// TIA Portal V20 export
DATA_BLOCK "Config"   // DB58
{ DB_Accessible_From_OPC_UA := 'FALSE' }
AUTHOR : ERsystem_FA2_DH. Kim
// stored: Access Published, DBAccessibleFromOPCUA false, DBAccessibleFromWebserver false, MemoryReserve 100, Namespace Unit1.Em6
   VAR
      em { ExternalWritable := 'False'} : "LAF_typeEmConfiguration";
      axis { ExternalAccessible := 'False'; ExternalVisible := 'False'; ExternalWritable := 'False'} : Array[1.._.U1EM6_NO_OF_AXES] of DB_ANY;
      outputCam : Array[1.._.U1EM6_NO_OF_OUTPUTCAM] of DB_ANY;
      cmStackTableElectrodeDetect { S7_SetPoint := 'True'} : "LBC_typeDigitalSignalConfiguration";
   END_VAR
   VAR RETAIN
      cmMasterVirtualAxisX { ExternalVisible := 'False'; ExternalWritable := 'False'} : "LBC_typeAxis64PosConfiguration";
      cmFinalRollerFrontAxisX { ExternalVisible := 'False'; ExternalWritable := 'False'} : "LBC_typeAxis64PosConfiguration";
      cmFinalRollerRearAxisX { ExternalVisible := 'False'; ExternalWritable := 'False'; S7_SetPoint := 'True'} : "LBC_typeAxis64PosConfiguration";
      cmMendrelAnodeFrontAxisY { ExternalVisible := 'False'; ExternalWritable := 'False'; S7_SetPoint := 'True'} : "LBC_typeAxis64PosConfiguration";
      cmMendrelAnodeFrontAxisZ { ExternalVisible := 'False'; ExternalWritable := 'False'; S7_SetPoint := 'True'} : "LBC_typeAxis64PosConfiguration";
      cmMendrelAnodeRearAxisY { ExternalVisible := 'False'; ExternalWritable := 'False'; S7_SetPoint := 'True'} : "LBC_typeAxis64PosConfiguration";
      cmMendrelAnodeRearAxisZ { ExternalVisible := 'False'; ExternalWritable := 'False'; S7_SetPoint := 'True'} : "LBC_typeAxis64PosConfiguration";
      cmMendrelCathodeFrontAxisY { ExternalVisible := 'False'; ExternalWritable := 'False'; S7_SetPoint := 'True'} : "LBC_typeAxis64PosConfiguration";
      cmMendrelCathodeFrontAxisZ { ExternalVisible := 'False'; ExternalWritable := 'False'; S7_SetPoint := 'True'} : "LBC_typeAxis64PosConfiguration";
      cmMendrelCathodeRearAxisY { ExternalVisible := 'False'; ExternalWritable := 'False'; S7_SetPoint := 'True'} : "LBC_typeAxis64PosConfiguration";
      cmMendrelCathodeRearAxisZ { ExternalVisible := 'False'; ExternalWritable := 'False'; S7_SetPoint := 'True'} : "LBC_typeAxis64PosConfiguration";
      cmStackTableAxisZ { ExternalVisible := 'False'; ExternalWritable := 'False'; S7_SetPoint := 'True'} : "LBC_typeAxis64PosConfiguration";
      cmStackTableOutFrontAxisZ { ExternalVisible := 'False'; ExternalWritable := 'False'; S7_SetPoint := 'True'} : "LBC_typeAxis64PosConfiguration";
      cmStackTableOutRearAxisZ { ExternalVisible := 'False'; ExternalWritable := 'False'; S7_SetPoint := 'True'} : "LBC_typeAxis64PosConfiguration";
   END_VAR
   VAR
      cmMendrelAnodeFrontClamp { ExternalAccessible := 'False'; ExternalVisible := 'False'; ExternalWritable := 'False'; S7_SetPoint := 'True'} : "LBC_typeTwoWayActuatorConfiguration";
      cmMendrelAnodeRearClamp { ExternalAccessible := 'False'; ExternalVisible := 'False'; ExternalWritable := 'False'; S7_SetPoint := 'True'} : "LBC_typeTwoWayActuatorConfiguration";
      cmMendrelCathodeFrontClamp { ExternalAccessible := 'False'; ExternalVisible := 'False'; ExternalWritable := 'False'; S7_SetPoint := 'True'} : "LBC_typeTwoWayActuatorConfiguration";
      cmMendrelCathodeRearClamp { ExternalAccessible := 'False'; ExternalVisible := 'False'; ExternalWritable := 'False'; S7_SetPoint := 'True'} : "LBC_typeTwoWayActuatorConfiguration";
      cmStackTableVaccum { ExternalAccessible := 'False'; ExternalVisible := 'False'; ExternalWritable := 'False'; S7_SetPoint := 'True'} : "LBC_typeTwoWayActuatorConfiguration";
      cmStackTableGapPadUpDown { ExternalAccessible := 'False'; ExternalVisible := 'False'; ExternalWritable := 'False'; S7_SetPoint := 'True'} : "LBC_typeTwoWayActuatorConfiguration";
      cmStackGapVisionControllerInterface { ExternalAccessible := 'False'; ExternalVisible := 'False'; ExternalWritable := 'False'; S7_SetPoint := 'True'} : "LER_typeVisionConfiguration";
   END_VAR
   VAR RETAIN
      softCam : Struct
         cmFinalRollerFrontAxisX : "LER_typeSoftCamInterface";
         cmFinalRollerRearAxisX { S7_SetPoint := 'True'} : "LER_typeSoftCamInterface";
         cmMendrelAnodeFrontAxisY { S7_SetPoint := 'True'} : "LER_typeSoftCamInterface";
         cmMendrelAnodeFrontAxisZ { S7_SetPoint := 'True'} : "LER_typeSoftCamInterface";
         cmMendrelAnodeRearAxisY { S7_SetPoint := 'True'} : "LER_typeSoftCamInterface";
         cmMendrelAnodeRearAxisZ { S7_SetPoint := 'True'} : "LER_typeSoftCamInterface";
         cmMendrelCathodeFrontAxisY { S7_SetPoint := 'True'} : "LER_typeSoftCamInterface";
         cmMendrelCathodeFrontAxisZ { S7_SetPoint := 'True'} : "LER_typeSoftCamInterface";
         cmMendrelCathodeRearAxisY { S7_SetPoint := 'True'} : "LER_typeSoftCamInterface";
         cmMendrelCathodeRearAxisZ { S7_SetPoint := 'True'} : "LER_typeSoftCamInterface";
         cmStackTableAxisZ { S7_SetPoint := 'True'} : "LER_typeSoftCamInterface";
         cmStackTableOutFrontAxisZ { S7_SetPoint := 'True'} : "LER_typeSoftCamInterface";
         cmStackTableOutRearAxisZ { S7_SetPoint := 'True'} : "LER_typeSoftCamInterface";
      END_STRUCT;
   END_VAR
BEGIN
   em.referenceDesignator.parent := WSTRING#'';
   em.referenceDesignator.relative := WSTRING#'';
   em.referenceDesignator.combined := WSTRING#'';
   axis[1] := 171;   // FinalRollerFrontAxisX
   axis[2] := 172;   // FinalRollerRearAxisX
   axis[3] := 163;   // MendrelAnodeFrontAxisY
   axis[4] := 162;   // MendrelAnodeFrontAxisZ
   axis[5] := 167;   // MendrelAnodeRearAxisY
   axis[6] := 166;   // MendrelAnodeRearAxisZ
   axis[7] := 161;   // MendrelCathodeFrontAxisY
   axis[8] := 160;   // MendrelCathodeFrontAxisZ
   axis[9] := 165;   // MendrelCathodeRearAxisY
   axis[10] := 164;   // MendrelCathodeRearAxisZ
   axis[11] := 168;   // StackTableAxisZ
   axis[12] := 169;   // StackTableOutFrontAxisZ
   axis[13] := 170;   // StackTableOutRearAxisZ
   axis[14] := 85;
   outputCam[1] := 224;
   outputCam[2] := 225;
   outputCam[3] := 206;
   outputCam[4] := 446;
   outputCam[5] := 445;
   outputCam[6] := 84;
   cmStackTableElectrodeDetect.referenceDesignator := WSTRING#'DigitalSignal';
   cmStackTableElectrodeDetect.onDelay := T#0MS;
   cmStackTableElectrodeDetect.offDelay := T#0MS;
   cmStackTableElectrodeDetect.default := FALSE;
   cmStackTableElectrodeDetect.invertProcessValue := FALSE;
   cmStackTableElectrodeDetect.disableAlarms := FALSE;
   cmMasterVirtualAxisX.referenceDesignator := WSTRING#'FinalRollerFrontAxisX';
   cmMasterVirtualAxisX.disableAlarms := FALSE;
   cmMasterVirtualAxisX.masterControlPopUp := TRUE;
   cmMasterVirtualAxisX.setPositions[0..15].position := 0.0;
   cmMasterVirtualAxisX.setPositions[0..15].velocity := -1.0;
   cmMasterVirtualAxisX.setPositions[0..15].acceleration := -1.0;
   cmMasterVirtualAxisX.setPositions[0..15].deceleration := -1.0;
   cmMasterVirtualAxisX.setPositions[0..15]."name" := '';
   cmFinalRollerFrontAxisX.referenceDesignator := WSTRING#'FinalRollerFrontAxisX';
   cmFinalRollerFrontAxisX.disableAlarms := FALSE;
   cmFinalRollerFrontAxisX.masterControlPopUp := TRUE;
   cmFinalRollerFrontAxisX.setPositions[0].position := 0.0;
   cmFinalRollerFrontAxisX.setPositions[1].position := 310.0;
   cmFinalRollerFrontAxisX.setPositions[2..15].position := 0.0;
   cmFinalRollerFrontAxisX.setPositions[0..1].velocity := 500.0;
   cmFinalRollerFrontAxisX.setPositions[2..3].velocity := 16#7FF8_0000_0000_0000;
   cmFinalRollerFrontAxisX.setPositions[4..15].velocity := -1.0;
   cmFinalRollerFrontAxisX.setPositions[0..1].acceleration := 5000.0;
   cmFinalRollerFrontAxisX.setPositions[2..3].acceleration := 16#7FF8_0000_0000_0000;
   cmFinalRollerFrontAxisX.setPositions[4..15].acceleration := -1.0;
   cmFinalRollerFrontAxisX.setPositions[0..1].deceleration := 5000.0;
   cmFinalRollerFrontAxisX.setPositions[2..3].deceleration := 16#7FF8_0000_0000_0000;
   cmFinalRollerFrontAxisX.setPositions[4..15].deceleration := -1.0;
   cmFinalRollerFrontAxisX.setPositions[0..15]."name" := '';
   cmFinalRollerRearAxisX.referenceDesignator := WSTRING#'FinalRollerRearAxisX';
   cmFinalRollerRearAxisX.disableAlarms := FALSE;
   cmFinalRollerRearAxisX.masterControlPopUp := TRUE;
   cmFinalRollerRearAxisX.setPositions[0].position := 0.0;
   cmFinalRollerRearAxisX.setPositions[1].position := 310.0;
   cmFinalRollerRearAxisX.setPositions[2..15].position := 0.0;
   cmFinalRollerRearAxisX.setPositions[0..1].velocity := 500.0;
   cmFinalRollerRearAxisX.setPositions[2..3].velocity := 16#7FF8_0000_0000_0000;
   cmFinalRollerRearAxisX.setPositions[4..15].velocity := -1.0;
   cmFinalRollerRearAxisX.setPositions[0..1].acceleration := 5000.0;
   cmFinalRollerRearAxisX.setPositions[2..3].acceleration := 16#7FF8_0000_0000_0000;
   cmFinalRollerRearAxisX.setPositions[4..15].acceleration := -1.0;
   cmFinalRollerRearAxisX.setPositions[0..1].deceleration := 5000.0;
   cmFinalRollerRearAxisX.setPositions[2..3].deceleration := 16#7FF8_0000_0000_0000;
   cmFinalRollerRearAxisX.setPositions[4..15].deceleration := -1.0;
   cmFinalRollerRearAxisX.setPositions[0..15]."name" := '';
   cmMendrelAnodeFrontAxisY.referenceDesignator := WSTRING#'MendrelAnodeFrontAxisY';
   cmMendrelAnodeFrontAxisY.disableAlarms := FALSE;
   cmMendrelAnodeFrontAxisY.masterControlPopUp := TRUE;
   cmMendrelAnodeFrontAxisY.setPositions[0].position := 0.0;
   cmMendrelAnodeFrontAxisY.setPositions[1].position := 50.0;
   cmMendrelAnodeFrontAxisY.setPositions[2..15].position := 0.0;
   cmMendrelAnodeFrontAxisY.setPositions[0..1].velocity := 50.0;
   cmMendrelAnodeFrontAxisY.setPositions[2..15].velocity := -1.0;
   cmMendrelAnodeFrontAxisY.setPositions[0..1].acceleration := 500.0;
   cmMendrelAnodeFrontAxisY.setPositions[2..15].acceleration := -1.0;
   cmMendrelAnodeFrontAxisY.setPositions[0..1].deceleration := 500.0;
   cmMendrelAnodeFrontAxisY.setPositions[2..15].deceleration := -1.0;
   cmMendrelAnodeFrontAxisY.setPositions[0..15]."name" := '';
   cmMendrelAnodeFrontAxisZ.referenceDesignator := WSTRING#'MendrelAnodeFrontAxisZ';
   cmMendrelAnodeFrontAxisZ.disableAlarms := FALSE;
   cmMendrelAnodeFrontAxisZ.masterControlPopUp := TRUE;
   cmMendrelAnodeFrontAxisZ.setPositions[0].position := 0.0;
   cmMendrelAnodeFrontAxisZ.setPositions[1].position := 50.0;
   cmMendrelAnodeFrontAxisZ.setPositions[2..15].position := 0.0;
   cmMendrelAnodeFrontAxisZ.setPositions[0..1].velocity := 50.0;
   cmMendrelAnodeFrontAxisZ.setPositions[2..15].velocity := -1.0;
   cmMendrelAnodeFrontAxisZ.setPositions[0..1].acceleration := 500.0;
   cmMendrelAnodeFrontAxisZ.setPositions[2..15].acceleration := -1.0;
   cmMendrelAnodeFrontAxisZ.setPositions[0..1].deceleration := 500.0;
   cmMendrelAnodeFrontAxisZ.setPositions[2..15].deceleration := -1.0;
   cmMendrelAnodeFrontAxisZ.setPositions[0..15]."name" := '';
   cmMendrelAnodeRearAxisY.referenceDesignator := WSTRING#'MendrelAnodeRearAxisY';
   cmMendrelAnodeRearAxisY.disableAlarms := FALSE;
   cmMendrelAnodeRearAxisY.masterControlPopUp := TRUE;
   cmMendrelAnodeRearAxisY.setPositions[0].position := 0.0;
   cmMendrelAnodeRearAxisY.setPositions[1].position := 50.0;
   cmMendrelAnodeRearAxisY.setPositions[2..15].position := 0.0;
   cmMendrelAnodeRearAxisY.setPositions[0..1].velocity := 50.0;
   cmMendrelAnodeRearAxisY.setPositions[2..15].velocity := -1.0;
   cmMendrelAnodeRearAxisY.setPositions[0..1].acceleration := 500.0;
   cmMendrelAnodeRearAxisY.setPositions[2..15].acceleration := -1.0;
   cmMendrelAnodeRearAxisY.setPositions[0..1].deceleration := 500.0;
   cmMendrelAnodeRearAxisY.setPositions[2..15].deceleration := -1.0;
   cmMendrelAnodeRearAxisY.setPositions[0..15]."name" := '';
   cmMendrelAnodeRearAxisZ.referenceDesignator := WSTRING#'MendrelAnodeRearAxisZ';
   cmMendrelAnodeRearAxisZ.disableAlarms := FALSE;
   cmMendrelAnodeRearAxisZ.masterControlPopUp := TRUE;
   cmMendrelAnodeRearAxisZ.setPositions[0].position := 0.0;
   cmMendrelAnodeRearAxisZ.setPositions[1].position := 50.0;
   cmMendrelAnodeRearAxisZ.setPositions[2..15].position := 0.0;
   cmMendrelAnodeRearAxisZ.setPositions[0..1].velocity := 50.0;
   cmMendrelAnodeRearAxisZ.setPositions[2..15].velocity := -1.0;
   cmMendrelAnodeRearAxisZ.setPositions[0..1].acceleration := 500.0;
   cmMendrelAnodeRearAxisZ.setPositions[2..15].acceleration := -1.0;
   cmMendrelAnodeRearAxisZ.setPositions[0..1].deceleration := 500.0;
   cmMendrelAnodeRearAxisZ.setPositions[2..15].deceleration := -1.0;
   cmMendrelAnodeRearAxisZ.setPositions[0..15]."name" := '';
   cmMendrelCathodeFrontAxisY.referenceDesignator := WSTRING#'MendrelCathodeFrontAxisY';
   cmMendrelCathodeFrontAxisY.disableAlarms := FALSE;
   cmMendrelCathodeFrontAxisY.masterControlPopUp := TRUE;
   cmMendrelCathodeFrontAxisY.setPositions[0].position := 0.0;
   cmMendrelCathodeFrontAxisY.setPositions[1].position := 50.0;
   cmMendrelCathodeFrontAxisY.setPositions[2..15].position := 0.0;
   cmMendrelCathodeFrontAxisY.setPositions[0..1].velocity := 50.0;
   cmMendrelCathodeFrontAxisY.setPositions[2..15].velocity := -1.0;
   cmMendrelCathodeFrontAxisY.setPositions[0..1].acceleration := 500.0;
   cmMendrelCathodeFrontAxisY.setPositions[2..15].acceleration := -1.0;
   cmMendrelCathodeFrontAxisY.setPositions[0..1].deceleration := 500.0;
   cmMendrelCathodeFrontAxisY.setPositions[2..15].deceleration := -1.0;
   cmMendrelCathodeFrontAxisY.setPositions[0..15]."name" := '';
   cmMendrelCathodeFrontAxisZ.referenceDesignator := WSTRING#'MendrelCathodeFrontAxisZ';
   cmMendrelCathodeFrontAxisZ.disableAlarms := FALSE;
   cmMendrelCathodeFrontAxisZ.masterControlPopUp := TRUE;
   cmMendrelCathodeFrontAxisZ.setPositions[0].position := 0.0;
   cmMendrelCathodeFrontAxisZ.setPositions[1].position := 50.0;
   cmMendrelCathodeFrontAxisZ.setPositions[2..15].position := 0.0;
   cmMendrelCathodeFrontAxisZ.setPositions[0..1].velocity := 50.0;
   cmMendrelCathodeFrontAxisZ.setPositions[2..15].velocity := -1.0;
   cmMendrelCathodeFrontAxisZ.setPositions[0..1].acceleration := 500.0;
   cmMendrelCathodeFrontAxisZ.setPositions[2..15].acceleration := -1.0;
   cmMendrelCathodeFrontAxisZ.setPositions[0..1].deceleration := 500.0;
   cmMendrelCathodeFrontAxisZ.setPositions[2..15].deceleration := -1.0;
   cmMendrelCathodeFrontAxisZ.setPositions[0..15]."name" := '';
   cmMendrelCathodeRearAxisY.referenceDesignator := WSTRING#'MendrelCathodeRearAxisY';
   cmMendrelCathodeRearAxisY.disableAlarms := FALSE;
   cmMendrelCathodeRearAxisY.masterControlPopUp := TRUE;
   cmMendrelCathodeRearAxisY.setPositions[0].position := 0.0;
   cmMendrelCathodeRearAxisY.setPositions[1].position := 50.0;
   cmMendrelCathodeRearAxisY.setPositions[2..15].position := 0.0;
   cmMendrelCathodeRearAxisY.setPositions[0..1].velocity := 50.0;
   cmMendrelCathodeRearAxisY.setPositions[2..15].velocity := -1.0;
   cmMendrelCathodeRearAxisY.setPositions[0..1].acceleration := 500.0;
   cmMendrelCathodeRearAxisY.setPositions[2..15].acceleration := -1.0;
   cmMendrelCathodeRearAxisY.setPositions[0..1].deceleration := 500.0;
   cmMendrelCathodeRearAxisY.setPositions[2..15].deceleration := -1.0;
   cmMendrelCathodeRearAxisY.setPositions[0..15]."name" := '';
   cmMendrelCathodeRearAxisZ.referenceDesignator := WSTRING#'MendrelCathodeRearAxisZ';
   cmMendrelCathodeRearAxisZ.disableAlarms := FALSE;
   cmMendrelCathodeRearAxisZ.masterControlPopUp := TRUE;
   cmMendrelCathodeRearAxisZ.setPositions[0].position := 0.0;
   cmMendrelCathodeRearAxisZ.setPositions[1].position := 50.0;
   cmMendrelCathodeRearAxisZ.setPositions[2..15].position := 0.0;
   cmMendrelCathodeRearAxisZ.setPositions[0..1].velocity := 50.0;
   cmMendrelCathodeRearAxisZ.setPositions[2..15].velocity := -1.0;
   cmMendrelCathodeRearAxisZ.setPositions[0..1].acceleration := 500.0;
   cmMendrelCathodeRearAxisZ.setPositions[2..15].acceleration := -1.0;
   cmMendrelCathodeRearAxisZ.setPositions[0..1].deceleration := 500.0;
   cmMendrelCathodeRearAxisZ.setPositions[2..15].deceleration := -1.0;
   cmMendrelCathodeRearAxisZ.setPositions[0..15]."name" := '';
   cmStackTableAxisZ.referenceDesignator := WSTRING#'StackTableAxisZ';
   cmStackTableAxisZ.disableAlarms := FALSE;
   cmStackTableAxisZ.masterControlPopUp := TRUE;
   cmStackTableAxisZ.setPositions[0].position := 0.0;
   cmStackTableAxisZ.setPositions[1].position := 5.0;
   cmStackTableAxisZ.setPositions[2..15].position := 0.0;
   cmStackTableAxisZ.setPositions[0..1].velocity := 50.0;
   cmStackTableAxisZ.setPositions[2..15].velocity := -1.0;
   cmStackTableAxisZ.setPositions[0..1].acceleration := 500.0;
   cmStackTableAxisZ.setPositions[2..15].acceleration := -1.0;
   cmStackTableAxisZ.setPositions[0..1].deceleration := 500.0;
   cmStackTableAxisZ.setPositions[2..15].deceleration := -1.0;
   cmStackTableAxisZ.setPositions[0..15]."name" := '';
   cmStackTableOutFrontAxisZ.referenceDesignator := WSTRING#'StackTableOutFrontAxisZ';
   cmStackTableOutFrontAxisZ.disableAlarms := FALSE;
   cmStackTableOutFrontAxisZ.masterControlPopUp := TRUE;
   cmStackTableOutFrontAxisZ.setPositions[0].position := 0.0;
   cmStackTableOutFrontAxisZ.setPositions[1].position := 500.0;
   cmStackTableOutFrontAxisZ.setPositions[2..15].position := 0.0;
   cmStackTableOutFrontAxisZ.setPositions[0..1].velocity := 500.0;
   cmStackTableOutFrontAxisZ.setPositions[2..15].velocity := -1.0;
   cmStackTableOutFrontAxisZ.setPositions[0..1].acceleration := 5000.0;
   cmStackTableOutFrontAxisZ.setPositions[2..15].acceleration := -1.0;
   cmStackTableOutFrontAxisZ.setPositions[0..1].deceleration := 5000.0;
   cmStackTableOutFrontAxisZ.setPositions[2..15].deceleration := -1.0;
   cmStackTableOutFrontAxisZ.setPositions[0..15]."name" := '';
   cmStackTableOutRearAxisZ.referenceDesignator := WSTRING#'StackTableOutRearAxisZ';
   cmStackTableOutRearAxisZ.disableAlarms := FALSE;
   cmStackTableOutRearAxisZ.masterControlPopUp := TRUE;
   cmStackTableOutRearAxisZ.setPositions[0].position := 0.0;
   cmStackTableOutRearAxisZ.setPositions[1].position := 500.0;
   cmStackTableOutRearAxisZ.setPositions[2..15].position := 0.0;
   cmStackTableOutRearAxisZ.setPositions[0..1].velocity := 500.0;
   cmStackTableOutRearAxisZ.setPositions[2..15].velocity := -1.0;
   cmStackTableOutRearAxisZ.setPositions[0..1].acceleration := 5000.0;
   cmStackTableOutRearAxisZ.setPositions[2..15].acceleration := -1.0;
   cmStackTableOutRearAxisZ.setPositions[0..1].deceleration := 5000.0;
   cmStackTableOutRearAxisZ.setPositions[2..15].deceleration := -1.0;
   cmStackTableOutRearAxisZ.setPositions[0..15]."name" := '';
   cmMendrelAnodeFrontClamp.referenceDesignator := WSTRING#'MendrelAnodeFrontClamp';
   cmMendrelAnodeRearClamp.referenceDesignator := WSTRING#'MendrelAnodeRearClamp';
   cmMendrelCathodeFrontClamp.referenceDesignator := WSTRING#'MendrelCathodeFrontClamp';
   cmMendrelCathodeRearClamp.referenceDesignator := WSTRING#'MendrelCathodeRearClamp';
   cmStackTableVaccum.referenceDesignator := WSTRING#'StackTableVaccum';
   cmStackTableVaccum.monitoringLeavingFeedback := T#5S;
   cmStackTableVaccum.monitoringReachingFeedback := T#5S;
   cmStackTableVaccum.monitoringDiscrepancy := T#0MS;
   cmStackTableVaccum.setOutputHomeContinuously := TRUE;
   cmStackTableVaccum.setOutputWorkContinuously := TRUE;
   cmStackTableVaccum.disableHomeCommand := FALSE;
   cmStackTableVaccum.disableFeedbackHomePos := FALSE;
   cmStackTableVaccum.disableFeedbackWorkPos := FALSE;
   cmStackTableVaccum.disableAlarms := FALSE;
   cmStackTableVaccum.resetOutputsOnError := FALSE;
   cmStackTableVaccum.allwaysWaitOnReachingTime := FALSE;
   cmStackTableGapPadUpDown.referenceDesignator := WSTRING#'StackTableGapPadUpDown';
   cmStackTableGapPadUpDown.monitoringLeavingFeedback := T#5S;
   cmStackTableGapPadUpDown.monitoringReachingFeedback := T#5S;
   cmStackTableGapPadUpDown.monitoringDiscrepancy := T#0MS;
   cmStackTableGapPadUpDown.setOutputHomeContinuously := TRUE;
   cmStackTableGapPadUpDown.setOutputWorkContinuously := TRUE;
   cmStackTableGapPadUpDown.disableHomeCommand := FALSE;
   cmStackTableGapPadUpDown.disableFeedbackHomePos := FALSE;
   cmStackTableGapPadUpDown.disableFeedbackWorkPos := FALSE;
   cmStackTableGapPadUpDown.disableAlarms := FALSE;
   cmStackTableGapPadUpDown.resetOutputsOnError := FALSE;
   cmStackTableGapPadUpDown.allwaysWaitOnReachingTime := FALSE;
   cmStackGapVisionControllerInterface.hwID.cmdResultStatusID := 463;
   cmStackGapVisionControllerInterface.hwID.trgReadyStatusID := 464;
   cmStackGapVisionControllerInterface.hwID.trgAckStatusID := 465;
   cmStackGapVisionControllerInterface.hwID.miscellaneousStatusID := 466;
   cmStackGapVisionControllerInterface.hwID.assignableStatusID := 467;
   cmStackGapVisionControllerInterface.hwID.resultData248ByteID_1 := 468;
   cmStackGapVisionControllerInterface.hwID.resultData248ByteID_2 := 893;
   cmStackGapVisionControllerInterface.hwID.resultData248ByteID_3 := 894;
   cmStackGapVisionControllerInterface.hwID.resultData248ByteID_4 := 895;
   cmStackGapVisionControllerInterface.hwID.resultData248ByteID_5 := 896;
   cmStackGapVisionControllerInterface.hwID.cmdResultControlID := 469;
   cmStackGapVisionControllerInterface.hwID.trgControlID := 470;
   cmStackGapVisionControllerInterface.hwID.miscellaneousControlID := 471;
   cmStackGapVisionControllerInterface.hwID.reservedControlID := 708;
   cmStackGapVisionControllerInterface.hwID.assignableControlID := 709;
   cmStackGapVisionControllerInterface.hwID.parameterData248ByteID_1 := 710;
   cmStackGapVisionControllerInterface.hwID.parameterData248ByteID_2 := 897;
   cmStackGapVisionControllerInterface.hwID.parameterData248ByteID_3 := 898;
   cmStackGapVisionControllerInterface.hwID.parameterData248ByteID_4 := 899;
   cmStackGapVisionControllerInterface.hwID.parameterData248ByteID_5 := 908;
   cmStackGapVisionControllerInterface.referenceDesignator := WSTRING#'StackGapVision';
   cmStackGapVisionControllerInterface.disableAlarms := FALSE;
   cmStackGapVisionControllerInterface.trigger1Use := FALSE;
   cmStackGapVisionControllerInterface.trigger2Use := FALSE;
   cmStackGapVisionControllerInterface.trigger3Use := FALSE;
   cmStackGapVisionControllerInterface.trigger4Use := FALSE;
   cmStackGapVisionControllerInterface.triggertime := T#0MS;
   cmStackGapVisionControllerInterface.cycleTime := T#0MS;
   cmStackGapVisionControllerInterface.DataConfig.cmdResultControl.cmdRequest := FALSE;
   cmStackGapVisionControllerInterface.DataConfig.cmdResultControl.inDataFbSyncInhibit := FALSE;
   cmStackGapVisionControllerInterface.DataConfig.cmdResultControl.reserved := FALSE;
   cmStackGapVisionControllerInterface.DataConfig.cmdResultControl.resultAck := FALSE;
   cmStackGapVisionControllerInterface.DataConfig.cmdResultControl.err0ResetRequest := FALSE;
   cmStackGapVisionControllerInterface.DataConfig.cmdResultControl.err1ResetRequest := FALSE;
   cmStackGapVisionControllerInterface.DataConfig.cmdResultControl.reserved0 := FALSE;
   cmStackGapVisionControllerInterface.DataConfig.cmdResultControl.reserved1 := FALSE;
   cmStackGapVisionControllerInterface.DataConfig.trgControl.trg1 := FALSE;
   cmStackGapVisionControllerInterface.DataConfig.trgControl.trg2 := FALSE;
   cmStackGapVisionControllerInterface.DataConfig.trgControl.trg3 := FALSE;
   cmStackGapVisionControllerInterface.DataConfig.trgControl.trg4 := FALSE;
   cmStackGapVisionControllerInterface.DataConfig.trgControl.reserved0 := FALSE;
   cmStackGapVisionControllerInterface.DataConfig.trgControl.reserved1 := FALSE;
   cmStackGapVisionControllerInterface.DataConfig.trgControl.reserved2 := FALSE;
   cmStackGapVisionControllerInterface.DataConfig.trgControl.reserved3 := FALSE;
   cmStackGapVisionControllerInterface.DataConfig.miscellaneousControl.reset := FALSE;
   cmStackGapVisionControllerInterface.DataConfig.miscellaneousControl.ext := FALSE;
   cmStackGapVisionControllerInterface.DataConfig.miscellaneousControl.test := FALSE;
   cmStackGapVisionControllerInterface.DataConfig.miscellaneousControl.reserved0 := FALSE;
   cmStackGapVisionControllerInterface.DataConfig.miscellaneousControl.reserved1 := FALSE;
   cmStackGapVisionControllerInterface.DataConfig.miscellaneousControl.reserved2 := FALSE;
   cmStackGapVisionControllerInterface.DataConfig.miscellaneousControl.reserved3 := FALSE;
   cmStackGapVisionControllerInterface.DataConfig.miscellaneousControl.reserved4 := FALSE;
   cmStackGapVisionControllerInterface.DataConfig.reservedControl.reserved0 := FALSE;
   cmStackGapVisionControllerInterface.DataConfig.reservedControl.reserved1 := FALSE;
   cmStackGapVisionControllerInterface.DataConfig.reservedControl.reserved2 := FALSE;
   cmStackGapVisionControllerInterface.DataConfig.reservedControl.reserved3 := FALSE;
   cmStackGapVisionControllerInterface.DataConfig.reservedControl.reserved4 := FALSE;
   cmStackGapVisionControllerInterface.DataConfig.reservedControl.reserved5 := FALSE;
   cmStackGapVisionControllerInterface.DataConfig.reservedControl.reserved6 := FALSE;
   cmStackGapVisionControllerInterface.DataConfig.reservedControl.reserved7 := FALSE;
   cmStackGapVisionControllerInterface.DataConfig.assignableControl.assignable_0 := FALSE;
   cmStackGapVisionControllerInterface.DataConfig.assignableControl.assignable_1 := FALSE;
   cmStackGapVisionControllerInterface.DataConfig.assignableControl.assignable_2 := FALSE;
   cmStackGapVisionControllerInterface.DataConfig.assignableControl.assignable_3 := FALSE;
   cmStackGapVisionControllerInterface.DataConfig.assignableControl.assignable_4 := FALSE;
   cmStackGapVisionControllerInterface.DataConfig.assignableControl.assignable_5 := FALSE;
   cmStackGapVisionControllerInterface.DataConfig.assignableControl.assignable_6 := FALSE;
   cmStackGapVisionControllerInterface.DataConfig.assignableControl.assignable_7 := FALSE;
   cmStackGapVisionControllerInterface.DataConfig.assignableControl.assignable_8 := FALSE;
   cmStackGapVisionControllerInterface.DataConfig.assignableControl.assignable_9 := FALSE;
   cmStackGapVisionControllerInterface.DataConfig.assignableControl.assignable_10 := FALSE;
   cmStackGapVisionControllerInterface.DataConfig.assignableControl.assignable_11 := FALSE;
   cmStackGapVisionControllerInterface.DataConfig.assignableControl.assignable_12 := FALSE;
   cmStackGapVisionControllerInterface.DataConfig.assignableControl.assignable_13 := FALSE;
   cmStackGapVisionControllerInterface.DataConfig.assignableControl.assignable_14 := FALSE;
   cmStackGapVisionControllerInterface.DataConfig.assignableControl.assignable_15 := FALSE;
   cmStackGapVisionControllerInterface.DataConfig.assignableControl.assignable_16 := FALSE;
   cmStackGapVisionControllerInterface.DataConfig.assignableControl.assignable_17 := FALSE;
   cmStackGapVisionControllerInterface.DataConfig.assignableControl.assignable_18 := FALSE;
   cmStackGapVisionControllerInterface.DataConfig.assignableControl.assignable_19 := FALSE;
   cmStackGapVisionControllerInterface.DataConfig.assignableControl.assignable_20 := FALSE;
   cmStackGapVisionControllerInterface.DataConfig.assignableControl.assignable_21 := FALSE;
   cmStackGapVisionControllerInterface.DataConfig.assignableControl.assignable_22 := FALSE;
   cmStackGapVisionControllerInterface.DataConfig.assignableControl.assignable_23 := FALSE;
   cmStackGapVisionControllerInterface.DataConfig.assignableControl.assignable_24 := FALSE;
   cmStackGapVisionControllerInterface.DataConfig.assignableControl.assignable_25 := FALSE;
   cmStackGapVisionControllerInterface.DataConfig.assignableControl.assignable_26 := FALSE;
   cmStackGapVisionControllerInterface.DataConfig.assignableControl.assignable_27 := FALSE;
   cmStackGapVisionControllerInterface.DataConfig.assignableControl.assignable_28 := FALSE;
   cmStackGapVisionControllerInterface.DataConfig.assignableControl.assignable_29 := FALSE;
   cmStackGapVisionControllerInterface.DataConfig.assignableControl.assignable_30 := FALSE;
   cmStackGapVisionControllerInterface.DataConfig.assignableControl.assignable_31 := FALSE;
   cmStackGapVisionControllerInterface.DataConfig.parameterData248Byte_1.reversed0 := 0;
   cmStackGapVisionControllerInterface.DataConfig.parameterData248Byte_1.reserved1 := 0;
   cmStackGapVisionControllerInterface.DataConfig.parameterData248Byte_1.commandNumber := 0;
   cmStackGapVisionControllerInterface.DataConfig.parameterData248Byte_1.cmdParameter[0..15] := 0;
   cmStackGapVisionControllerInterface.DataConfig.parameterData248Byte_1.inDataFieldbus[0..42] := 0;
   cmStackGapVisionControllerInterface.DataConfig.parameterData248Byte_2[0..61] := 0;
   cmStackGapVisionControllerInterface.DataConfig.parameterData248Byte_3[0..61] := 0;
   cmStackGapVisionControllerInterface.DataConfig.parameterData248Byte_4[0..61] := 0;
   cmStackGapVisionControllerInterface.DataConfig.parameterData248Byte_5[0..61] := 0;
   softCam.cmFinalRollerFrontAxisX.TargetPosition := 0.0;
   softCam.cmFinalRollerFrontAxisX.ActualPosition := 0.0;
   softCam.cmFinalRollerFrontAxisX.UnitName := WSTRING#'';
   softCam.cmFinalRollerFrontAxisX.error := FALSE;
   softCam.cmFinalRollerFrontAxisX.status := 16#0000;
   softCam.cmFinalRollerFrontAxisX.position[0..15].SetValue.Negative := 0.0;
   softCam.cmFinalRollerFrontAxisX.position[0..15].SetValue.Postive := 0.0;
   softCam.cmFinalRollerFrontAxisX.position[0..15].ProcessValue.Postive := 0.0;
   softCam.cmFinalRollerFrontAxisX.position[0..15].ProcessValue.Negative := 0.0;
   softCam.cmFinalRollerFrontAxisX.position[0..15].ProcessValue.SetPos := 0.0;
   softCam.cmFinalRollerFrontAxisX.position[0..15].ProcessValue.inPos := FALSE;
   softCam.cmFinalRollerFrontAxisX.position[0..15].ProcessValue.isBefore := FALSE;
   softCam.cmFinalRollerFrontAxisX.position[0..15].ProcessValue.isAfter := FALSE;
   softCam.cmFinalRollerFrontAxisX.position[0..15].ProcessValue.PosName := WSTRING#'';
   softCam.cmFinalRollerRearAxisX.TargetPosition := 0.0;
   softCam.cmFinalRollerRearAxisX.ActualPosition := 0.0;
   softCam.cmFinalRollerRearAxisX.UnitName := WSTRING#'';
   softCam.cmFinalRollerRearAxisX.error := FALSE;
   softCam.cmFinalRollerRearAxisX.status := 16#0000;
   softCam.cmFinalRollerRearAxisX.position[0..15].SetValue.Negative := 0.0;
   softCam.cmFinalRollerRearAxisX.position[0..15].SetValue.Postive := 0.0;
   softCam.cmFinalRollerRearAxisX.position[0..15].ProcessValue.Postive := 0.0;
   softCam.cmFinalRollerRearAxisX.position[0..15].ProcessValue.Negative := 0.0;
   softCam.cmFinalRollerRearAxisX.position[0..15].ProcessValue.SetPos := 0.0;
   softCam.cmFinalRollerRearAxisX.position[0..15].ProcessValue.inPos := FALSE;
   softCam.cmFinalRollerRearAxisX.position[0..15].ProcessValue.isBefore := FALSE;
   softCam.cmFinalRollerRearAxisX.position[0..15].ProcessValue.isAfter := FALSE;
   softCam.cmFinalRollerRearAxisX.position[0..15].ProcessValue.PosName := WSTRING#'';
   softCam.cmMendrelAnodeFrontAxisY.TargetPosition := 0.0;
   softCam.cmMendrelAnodeFrontAxisY.ActualPosition := 0.0;
   softCam.cmMendrelAnodeFrontAxisY.UnitName := WSTRING#'';
   softCam.cmMendrelAnodeFrontAxisY.error := FALSE;
   softCam.cmMendrelAnodeFrontAxisY.status := 16#0000;
   softCam.cmMendrelAnodeFrontAxisY.position[0..15].SetValue.Negative := 0.0;
   softCam.cmMendrelAnodeFrontAxisY.position[0..15].SetValue.Postive := 0.0;
   softCam.cmMendrelAnodeFrontAxisY.position[0..15].ProcessValue.Postive := 0.0;
   softCam.cmMendrelAnodeFrontAxisY.position[0..15].ProcessValue.Negative := 0.0;
   softCam.cmMendrelAnodeFrontAxisY.position[0..15].ProcessValue.SetPos := 0.0;
   softCam.cmMendrelAnodeFrontAxisY.position[0..15].ProcessValue.inPos := FALSE;
   softCam.cmMendrelAnodeFrontAxisY.position[0..15].ProcessValue.isBefore := FALSE;
   softCam.cmMendrelAnodeFrontAxisY.position[0..15].ProcessValue.isAfter := FALSE;
   softCam.cmMendrelAnodeFrontAxisY.position[0..15].ProcessValue.PosName := WSTRING#'';
   softCam.cmMendrelAnodeFrontAxisZ.TargetPosition := 0.0;
   softCam.cmMendrelAnodeFrontAxisZ.ActualPosition := 0.0;
   softCam.cmMendrelAnodeFrontAxisZ.UnitName := WSTRING#'';
   softCam.cmMendrelAnodeFrontAxisZ.error := FALSE;
   softCam.cmMendrelAnodeFrontAxisZ.status := 16#0000;
   softCam.cmMendrelAnodeFrontAxisZ.position[0..15].SetValue.Negative := 0.0;
   softCam.cmMendrelAnodeFrontAxisZ.position[0..15].SetValue.Postive := 0.0;
   softCam.cmMendrelAnodeFrontAxisZ.position[0..15].ProcessValue.Postive := 0.0;
   softCam.cmMendrelAnodeFrontAxisZ.position[0..15].ProcessValue.Negative := 0.0;
   softCam.cmMendrelAnodeFrontAxisZ.position[0..15].ProcessValue.SetPos := 0.0;
   softCam.cmMendrelAnodeFrontAxisZ.position[0..15].ProcessValue.inPos := FALSE;
   softCam.cmMendrelAnodeFrontAxisZ.position[0..15].ProcessValue.isBefore := FALSE;
   softCam.cmMendrelAnodeFrontAxisZ.position[0..15].ProcessValue.isAfter := FALSE;
   softCam.cmMendrelAnodeFrontAxisZ.position[0..15].ProcessValue.PosName := WSTRING#'';
   softCam.cmMendrelAnodeRearAxisY.TargetPosition := 0.0;
   softCam.cmMendrelAnodeRearAxisY.ActualPosition := 0.0;
   softCam.cmMendrelAnodeRearAxisY.UnitName := WSTRING#'';
   softCam.cmMendrelAnodeRearAxisY.error := FALSE;
   softCam.cmMendrelAnodeRearAxisY.status := 16#0000;
   softCam.cmMendrelAnodeRearAxisY.position[0..15].SetValue.Negative := 0.0;
   softCam.cmMendrelAnodeRearAxisY.position[0..15].SetValue.Postive := 0.0;
   softCam.cmMendrelAnodeRearAxisY.position[0..15].ProcessValue.Postive := 0.0;
   softCam.cmMendrelAnodeRearAxisY.position[0..15].ProcessValue.Negative := 0.0;
   softCam.cmMendrelAnodeRearAxisY.position[0..15].ProcessValue.SetPos := 0.0;
   softCam.cmMendrelAnodeRearAxisY.position[0..15].ProcessValue.inPos := FALSE;
   softCam.cmMendrelAnodeRearAxisY.position[0..15].ProcessValue.isBefore := FALSE;
   softCam.cmMendrelAnodeRearAxisY.position[0..15].ProcessValue.isAfter := FALSE;
   softCam.cmMendrelAnodeRearAxisY.position[0..15].ProcessValue.PosName := WSTRING#'';
   softCam.cmMendrelAnodeRearAxisZ.TargetPosition := 0.0;
   softCam.cmMendrelAnodeRearAxisZ.ActualPosition := 0.0;
   softCam.cmMendrelAnodeRearAxisZ.UnitName := WSTRING#'';
   softCam.cmMendrelAnodeRearAxisZ.error := FALSE;
   softCam.cmMendrelAnodeRearAxisZ.status := 16#0000;
   softCam.cmMendrelAnodeRearAxisZ.position[0..15].SetValue.Negative := 0.0;
   softCam.cmMendrelAnodeRearAxisZ.position[0..15].SetValue.Postive := 0.0;
   softCam.cmMendrelAnodeRearAxisZ.position[0..15].ProcessValue.Postive := 0.0;
   softCam.cmMendrelAnodeRearAxisZ.position[0..15].ProcessValue.Negative := 0.0;
   softCam.cmMendrelAnodeRearAxisZ.position[0..15].ProcessValue.SetPos := 0.0;
   softCam.cmMendrelAnodeRearAxisZ.position[0..15].ProcessValue.inPos := FALSE;
   softCam.cmMendrelAnodeRearAxisZ.position[0..15].ProcessValue.isBefore := FALSE;
   softCam.cmMendrelAnodeRearAxisZ.position[0..15].ProcessValue.isAfter := FALSE;
   softCam.cmMendrelAnodeRearAxisZ.position[0..15].ProcessValue.PosName := WSTRING#'';
   softCam.cmMendrelCathodeFrontAxisY.TargetPosition := 0.0;
   softCam.cmMendrelCathodeFrontAxisY.ActualPosition := 0.0;
   softCam.cmMendrelCathodeFrontAxisY.UnitName := WSTRING#'';
   softCam.cmMendrelCathodeFrontAxisY.error := FALSE;
   softCam.cmMendrelCathodeFrontAxisY.status := 16#0000;
   softCam.cmMendrelCathodeFrontAxisY.position[0..15].SetValue.Negative := 0.0;
   softCam.cmMendrelCathodeFrontAxisY.position[0..15].SetValue.Postive := 0.0;
   softCam.cmMendrelCathodeFrontAxisY.position[0..15].ProcessValue.Postive := 0.0;
   softCam.cmMendrelCathodeFrontAxisY.position[0..15].ProcessValue.Negative := 0.0;
   softCam.cmMendrelCathodeFrontAxisY.position[0..15].ProcessValue.SetPos := 0.0;
   softCam.cmMendrelCathodeFrontAxisY.position[0..15].ProcessValue.inPos := FALSE;
   softCam.cmMendrelCathodeFrontAxisY.position[0..15].ProcessValue.isBefore := FALSE;
   softCam.cmMendrelCathodeFrontAxisY.position[0..15].ProcessValue.isAfter := FALSE;
   softCam.cmMendrelCathodeFrontAxisY.position[0..15].ProcessValue.PosName := WSTRING#'';
   softCam.cmMendrelCathodeFrontAxisZ.TargetPosition := 0.0;
   softCam.cmMendrelCathodeFrontAxisZ.ActualPosition := 0.0;
   softCam.cmMendrelCathodeFrontAxisZ.UnitName := WSTRING#'';
   softCam.cmMendrelCathodeFrontAxisZ.error := FALSE;
   softCam.cmMendrelCathodeFrontAxisZ.status := 16#0000;
   softCam.cmMendrelCathodeFrontAxisZ.position[0..15].SetValue.Negative := 0.0;
   softCam.cmMendrelCathodeFrontAxisZ.position[0..15].SetValue.Postive := 0.0;
   softCam.cmMendrelCathodeFrontAxisZ.position[0..15].ProcessValue.Postive := 0.0;
   softCam.cmMendrelCathodeFrontAxisZ.position[0..15].ProcessValue.Negative := 0.0;
   softCam.cmMendrelCathodeFrontAxisZ.position[0..15].ProcessValue.SetPos := 0.0;
   softCam.cmMendrelCathodeFrontAxisZ.position[0..15].ProcessValue.inPos := FALSE;
   softCam.cmMendrelCathodeFrontAxisZ.position[0..15].ProcessValue.isBefore := FALSE;
   softCam.cmMendrelCathodeFrontAxisZ.position[0..15].ProcessValue.isAfter := FALSE;
   softCam.cmMendrelCathodeFrontAxisZ.position[0..15].ProcessValue.PosName := WSTRING#'';
   softCam.cmMendrelCathodeRearAxisY.TargetPosition := 0.0;
   softCam.cmMendrelCathodeRearAxisY.ActualPosition := 0.0;
   softCam.cmMendrelCathodeRearAxisY.UnitName := WSTRING#'';
   softCam.cmMendrelCathodeRearAxisY.error := FALSE;
   softCam.cmMendrelCathodeRearAxisY.status := 16#0000;
   softCam.cmMendrelCathodeRearAxisY.position[0..15].SetValue.Negative := 0.0;
   softCam.cmMendrelCathodeRearAxisY.position[0..15].SetValue.Postive := 0.0;
   softCam.cmMendrelCathodeRearAxisY.position[0..15].ProcessValue.Postive := 0.0;
   softCam.cmMendrelCathodeRearAxisY.position[0..15].ProcessValue.Negative := 0.0;
   softCam.cmMendrelCathodeRearAxisY.position[0..15].ProcessValue.SetPos := 0.0;
   softCam.cmMendrelCathodeRearAxisY.position[0..15].ProcessValue.inPos := FALSE;
   softCam.cmMendrelCathodeRearAxisY.position[0..15].ProcessValue.isBefore := FALSE;
   softCam.cmMendrelCathodeRearAxisY.position[0..15].ProcessValue.isAfter := FALSE;
   softCam.cmMendrelCathodeRearAxisY.position[0..15].ProcessValue.PosName := WSTRING#'';
   softCam.cmMendrelCathodeRearAxisZ.TargetPosition := 0.0;
   softCam.cmMendrelCathodeRearAxisZ.ActualPosition := 0.0;
   softCam.cmMendrelCathodeRearAxisZ.UnitName := WSTRING#'';
   softCam.cmMendrelCathodeRearAxisZ.error := FALSE;
   softCam.cmMendrelCathodeRearAxisZ.status := 16#0000;
   softCam.cmMendrelCathodeRearAxisZ.position[0..15].SetValue.Negative := 0.0;
   softCam.cmMendrelCathodeRearAxisZ.position[0..15].SetValue.Postive := 0.0;
   softCam.cmMendrelCathodeRearAxisZ.position[0..15].ProcessValue.Postive := 0.0;
   softCam.cmMendrelCathodeRearAxisZ.position[0..15].ProcessValue.Negative := 0.0;
   softCam.cmMendrelCathodeRearAxisZ.position[0..15].ProcessValue.SetPos := 0.0;
   softCam.cmMendrelCathodeRearAxisZ.position[0..15].ProcessValue.inPos := FALSE;
   softCam.cmMendrelCathodeRearAxisZ.position[0..15].ProcessValue.isBefore := FALSE;
   softCam.cmMendrelCathodeRearAxisZ.position[0..15].ProcessValue.isAfter := FALSE;
   softCam.cmMendrelCathodeRearAxisZ.position[0..15].ProcessValue.PosName := WSTRING#'';
   softCam.cmStackTableAxisZ.TargetPosition := 0.0;
   softCam.cmStackTableAxisZ.ActualPosition := 0.0;
   softCam.cmStackTableAxisZ.UnitName := WSTRING#'';
   softCam.cmStackTableAxisZ.error := FALSE;
   softCam.cmStackTableAxisZ.status := 16#0000;
   softCam.cmStackTableAxisZ.position[0..15].SetValue.Negative := 0.0;
   softCam.cmStackTableAxisZ.position[0..15].SetValue.Postive := 0.0;
   softCam.cmStackTableAxisZ.position[0..15].ProcessValue.Postive := 0.0;
   softCam.cmStackTableAxisZ.position[0..15].ProcessValue.Negative := 0.0;
   softCam.cmStackTableAxisZ.position[0..15].ProcessValue.SetPos := 0.0;
   softCam.cmStackTableAxisZ.position[0..15].ProcessValue.inPos := FALSE;
   softCam.cmStackTableAxisZ.position[0..15].ProcessValue.isBefore := FALSE;
   softCam.cmStackTableAxisZ.position[0..15].ProcessValue.isAfter := FALSE;
   softCam.cmStackTableAxisZ.position[0..15].ProcessValue.PosName := WSTRING#'';
   softCam.cmStackTableOutFrontAxisZ.TargetPosition := 0.0;
   softCam.cmStackTableOutFrontAxisZ.ActualPosition := 0.0;
   softCam.cmStackTableOutFrontAxisZ.UnitName := WSTRING#'';
   softCam.cmStackTableOutFrontAxisZ.error := FALSE;
   softCam.cmStackTableOutFrontAxisZ.status := 16#0000;
   softCam.cmStackTableOutFrontAxisZ.position[0..15].SetValue.Negative := 0.0;
   softCam.cmStackTableOutFrontAxisZ.position[0..15].SetValue.Postive := 0.0;
   softCam.cmStackTableOutFrontAxisZ.position[0..15].ProcessValue.Postive := 0.0;
   softCam.cmStackTableOutFrontAxisZ.position[0..15].ProcessValue.Negative := 0.0;
   softCam.cmStackTableOutFrontAxisZ.position[0..15].ProcessValue.SetPos := 0.0;
   softCam.cmStackTableOutFrontAxisZ.position[0..15].ProcessValue.inPos := FALSE;
   softCam.cmStackTableOutFrontAxisZ.position[0..15].ProcessValue.isBefore := FALSE;
   softCam.cmStackTableOutFrontAxisZ.position[0..15].ProcessValue.isAfter := FALSE;
   softCam.cmStackTableOutFrontAxisZ.position[0..15].ProcessValue.PosName := WSTRING#'';
   softCam.cmStackTableOutRearAxisZ.TargetPosition := 0.0;
   softCam.cmStackTableOutRearAxisZ.ActualPosition := 0.0;
   softCam.cmStackTableOutRearAxisZ.UnitName := WSTRING#'';
   softCam.cmStackTableOutRearAxisZ.error := FALSE;
   softCam.cmStackTableOutRearAxisZ.status := 16#0000;
   softCam.cmStackTableOutRearAxisZ.position[0..15].SetValue.Negative := 0.0;
   softCam.cmStackTableOutRearAxisZ.position[0..15].SetValue.Postive := 0.0;
   softCam.cmStackTableOutRearAxisZ.position[0..15].ProcessValue.Postive := 0.0;
   softCam.cmStackTableOutRearAxisZ.position[0..15].ProcessValue.Negative := 0.0;
   softCam.cmStackTableOutRearAxisZ.position[0..15].ProcessValue.SetPos := 0.0;
   softCam.cmStackTableOutRearAxisZ.position[0..15].ProcessValue.inPos := FALSE;
   softCam.cmStackTableOutRearAxisZ.position[0..15].ProcessValue.isBefore := FALSE;
   softCam.cmStackTableOutRearAxisZ.position[0..15].ProcessValue.isAfter := FALSE;
   softCam.cmStackTableOutRearAxisZ.position[0..15].ProcessValue.PosName := WSTRING#'';
END_DATA_BLOCK
